PROGRAM prgBattery
VAR
	byBatteryIslandOperation	: BOOL;							//{#lynus.ag#()}
	lrPowerBattery				: LREAL;						//{#lynus.ag#()}
	dwSOCBattery				: DWORD;						//{#lynus.ag#()}
	rTargetPowerBattery			: REAL;							//{#lynus.ag#()}
	bIsEnabledBattery			: BOOL;							//{#lynus.ag#()}
	bSResetBattery				: BOOL;							//{#lynus.ag#()}
	lrActualCapacityBattery		: LREAL;						//{#lynus.ag#()}
	lrMaxCapacityBattery		: LREAL;						//{#lynus.ag#()}
	byPrioBattery				: BYTE;							//{#lynus.ag#()}
	bEnableBattery				: BOOL;							//{#lynus.ag#()}
	bResetBattery				: BOOL;							//{#lynus.ag#()}


END_VAR

 prgBattery.lrPowerBattery					:=		prg_ADS.struct_received.lrPowerBattery			;
 prgBattery.dwSOCBattery					:=		prg_ADS.struct_received.dwSOCBattery			;
 prgBattery.rTargetPowerBattery				:=		prg_ADS.struct_received.rTargetPowerBattery			;
 prgBattery.bIsEnabledBattery				:=		prg_ADS.struct_received.bIsEnabledBattery			;
 prgBattery.bSResetBattery					:=		prg_ADS.struct_received.bSResetBattery			;
 prgBattery.lrActualCapacityBattery			:=		prg_ADS.struct_received.lrActualCapacityBattery			;
 prgBattery.lrMaxCapacityBattery			:=		prg_ADS.struct_received.lrMaxCapacityBattery			;
 prgBattery.byPrioBattery					:=		prg_ADS.struct_received.byPrioBattery			;
 prgBattery.bEnableBattery					:=		prg_ADS.struct_received.bEnableBattery			;
 prgBattery.bResetBattery					:=		prg_ADS.struct_received.bResetBattery			;

END_PROGRAM

(* stored: Version 1.1.0.1, ProductVersion 3.1.4024.12
   POU prgBattery: Id {a981e1b5-4989-4425-8d4d-bac69c77b6c8}, SpecialFunc None *)
